// Mitsubishi GX Works2 project: carwash_Q02H_v1   PLC: Q02/Q02H

PROGRAM MAIN
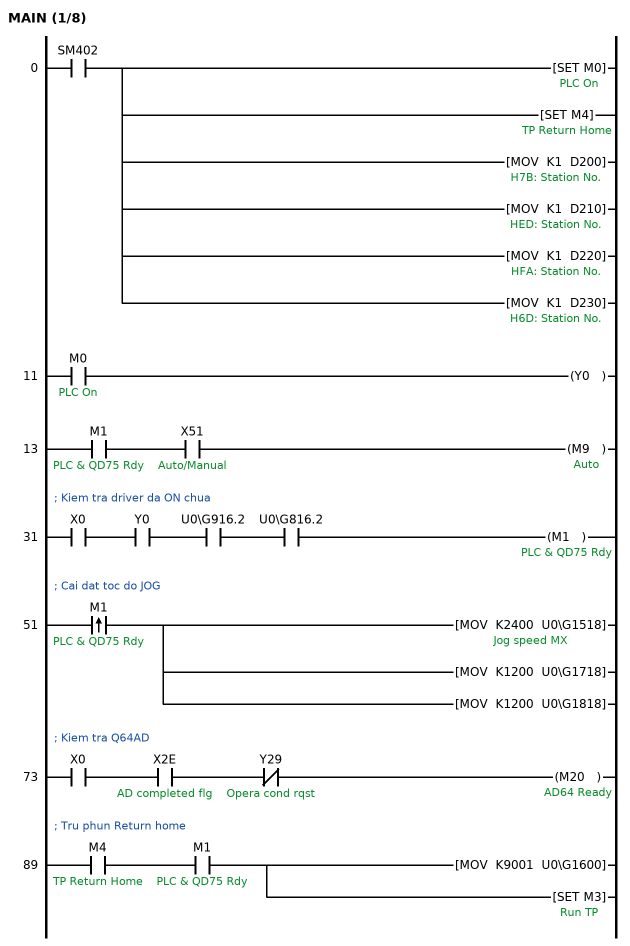
0     LD      SM402
      SET     M0  ; PLC On
      SET     M4  ; TP Return Home
      MOV     K1 D200  ; H7B: Station No.
      MOV     K1 D210  ; HED: Station No.
      MOV     K1 D220  ; HFA: Station No.
      MOV     K1 D230  ; H6D: Station No.
11    LD      M0  ; PLC On
      OUT     Y0
13    LD      M1  ; PLC & QD75 Rdy
      AND     X51  ; Auto/Manual
      OUT     M9  ; Auto
; Kiem tra driver da ON chua
31    LD      X0
      AND     Y0
      AND     U0\G916.2
      AND     U0\G816.2
      OUT     M1  ; PLC & QD75 Rdy
; Cai dat toc do JOG
51    LDP     M1  ; PLC & QD75 Rdy
      MOV     K2400 U0\G1518  ; Jog speed MX
      MOV     K1200 U0\G1718
      MOV     K1200 U0\G1818
; Kiem tra Q64AD
73    LD      X0
      AND     X2E  ; AD completed flg
      ANI     Y29  ; Opera cond rqst
      OUT     M20  ; AD64 Ready
; Tru phun Return home
89    LD      M4  ; TP Return Home
      AND     M1  ; PLC & QD75 Rdy
      MOV     K9001 U0\G1600
      SET     M3  ; Run TP
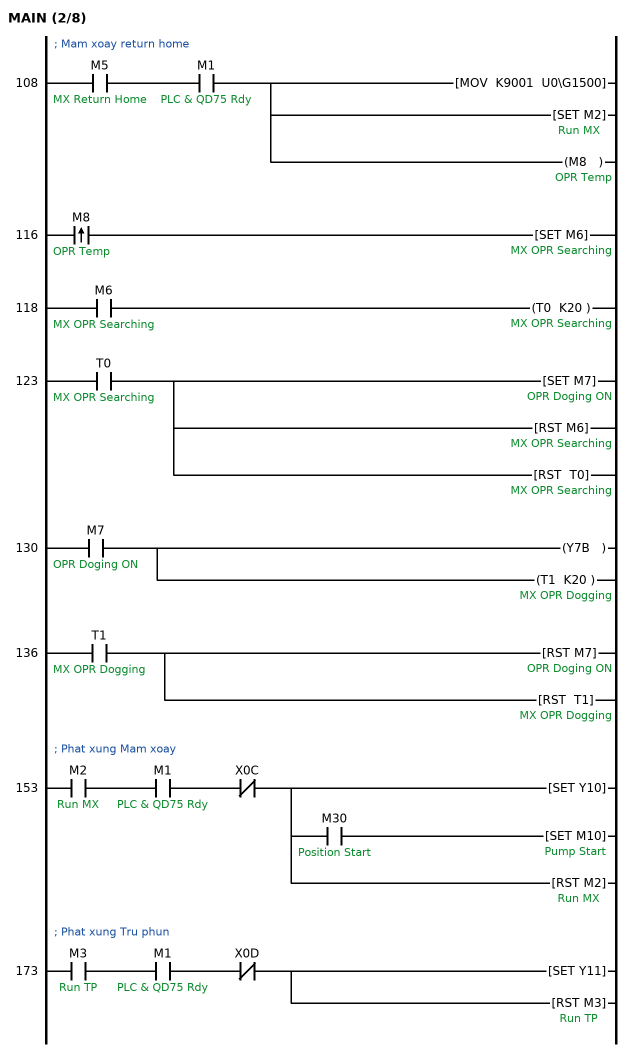
; Mam xoay return home
108   LD      M5  ; MX Return Home
      AND     M1  ; PLC & QD75 Rdy
      MOV     K9001 U0\G1500
      SET     M2  ; Run MX
      OUT     M8  ; OPR Temp
116   LDP     M8  ; OPR Temp
      SET     M6  ; MX OPR Searching
118   LD      M6  ; MX OPR Searching
      OUT     T0 K20  ; MX OPR Searching
123   LD      T0  ; MX OPR Searching
      SET     M7  ; OPR Doging ON
      RST     M6  ; MX OPR Searching
      RST     T0  ; MX OPR Searching
130   LD      M7  ; OPR Doging ON
      OUT     Y7B
      OUT     T1 K20  ; MX OPR Dogging
136   LD      T1  ; MX OPR Dogging
      RST     M7  ; OPR Doging ON
      RST     T1  ; MX OPR Dogging
; Phat xung Mam xoay
153   LD      M2  ; Run MX
      AND     M1  ; PLC & QD75 Rdy
      ANI     X0C
      SET     Y10
      MPS
      AND     M30  ; Position Start
      SET     M10  ; Pump Start
      MPP
      RST     M2  ; Run MX
; Phat xung Tru phun
173   LD      M3  ; Run TP
      AND     M1  ; PLC & QD75 Rdy
      ANI     X0D
      SET     Y11
      RST     M3  ; Run TP
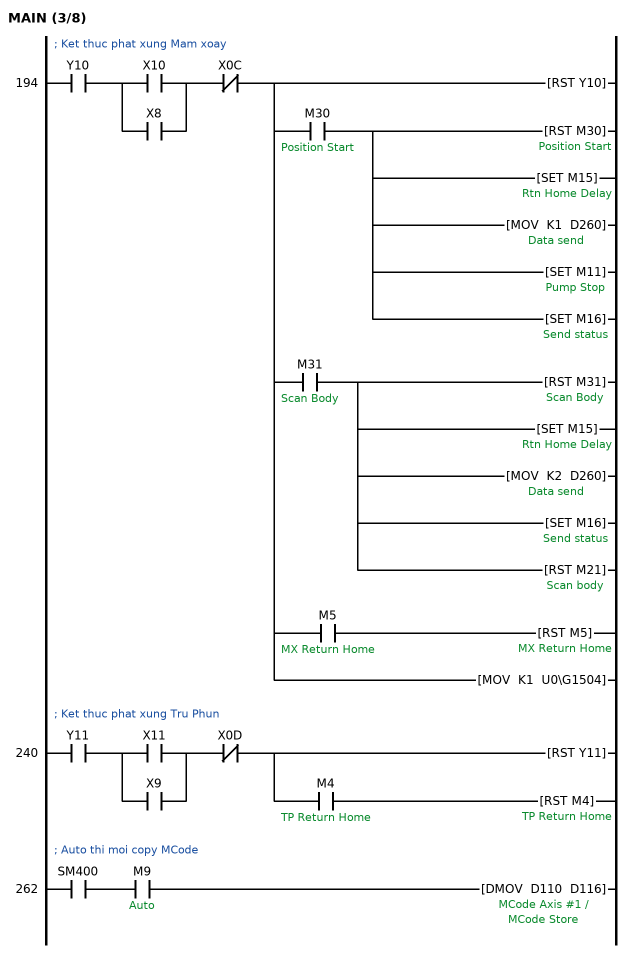
; Ket thuc phat xung Mam xoay
194   LD      Y10
      LD      X10
      OR      X8
      ANB
      ANI     X0C
      RST     Y10
      MPS
      AND     M30  ; Position Start
      RST     M30  ; Position Start
      SET     M15  ; Rtn Home Delay
      MOV     K1 D260  ; Data send
      SET     M11  ; Pump Stop
      SET     M16  ; Send status
      MRD
      AND     M31  ; Scan Body
      RST     M31  ; Scan Body
      SET     M15  ; Rtn Home Delay
      MOV     K2 D260
      SET     M16  ; Send status
      RST     M21  ; Scan body
      MRD
      AND     M5  ; MX Return Home
      RST     M5  ; MX Return Home
      MPP
      MOV     K1 U0\G1504
; Ket thuc phat xung Tru Phun
240   LD      Y11
      LD      X11
      OR      X9
      ANB
      ANI     X0D
      RST     Y11
      AND     M4  ; TP Return Home
      RST     M4  ; TP Return Home
; Auto thi moi copy MCode
262   LD      SM400
      AND     M9  ; Auto
      DMOV    D110 D116  ; MCode Axis #1 / MCode Store
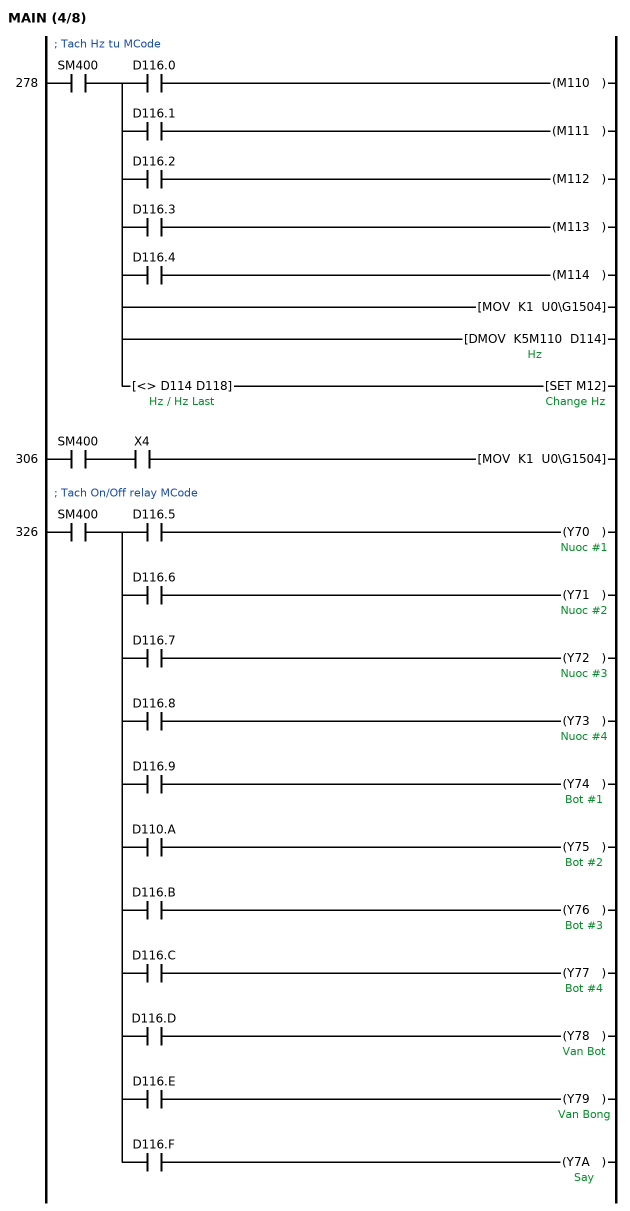
; Tach Hz tu MCode
278   LD      SM400
      MPS
      AND     D116.0
      OUT     M110
      MRD
      AND     D116.1
      OUT     M111
      MRD
      AND     D116.2
      OUT     M112
      MRD
      AND     D116.3
      OUT     M113
      MRD
      AND     D116.4
      OUT     M114
      MPP
      MOV     K1 U0\G1504
      DMOV    K5M110 D114  ; Hz
      AND<>   D114 D118  ; Hz / Hz Last
      SET     M12  ; Change Hz
306   LD      SM400
      AND     X4
      MOV     K1 U0\G1504
; Tach On/Off relay MCode
326   LD      SM400
      MPS
      AND     D116.5
      OUT     Y70  ; Nuoc #1
      MRD
      AND     D116.6
      OUT     Y71  ; Nuoc #2
      MRD
      AND     D116.7
      OUT     Y72  ; Nuoc #3
      MRD
      AND     D116.8
      OUT     Y73  ; Nuoc #4
      MRD
      AND     D116.9
      OUT     Y74  ; Bot #1
      MRD
      AND     D110.A
      OUT     Y75  ; Bot #2
      MRD
      AND     D116.B
      OUT     Y76  ; Bot #3
      MRD
      AND     D116.C
      OUT     Y77  ; Bot #4
      MRD
      AND     D116.D
      OUT     Y78  ; Van Bot
      MRD
      AND     D116.E
      OUT     Y79  ; Van Bong
      MPP
      AND     D116.F
      OUT     Y7A  ; Say
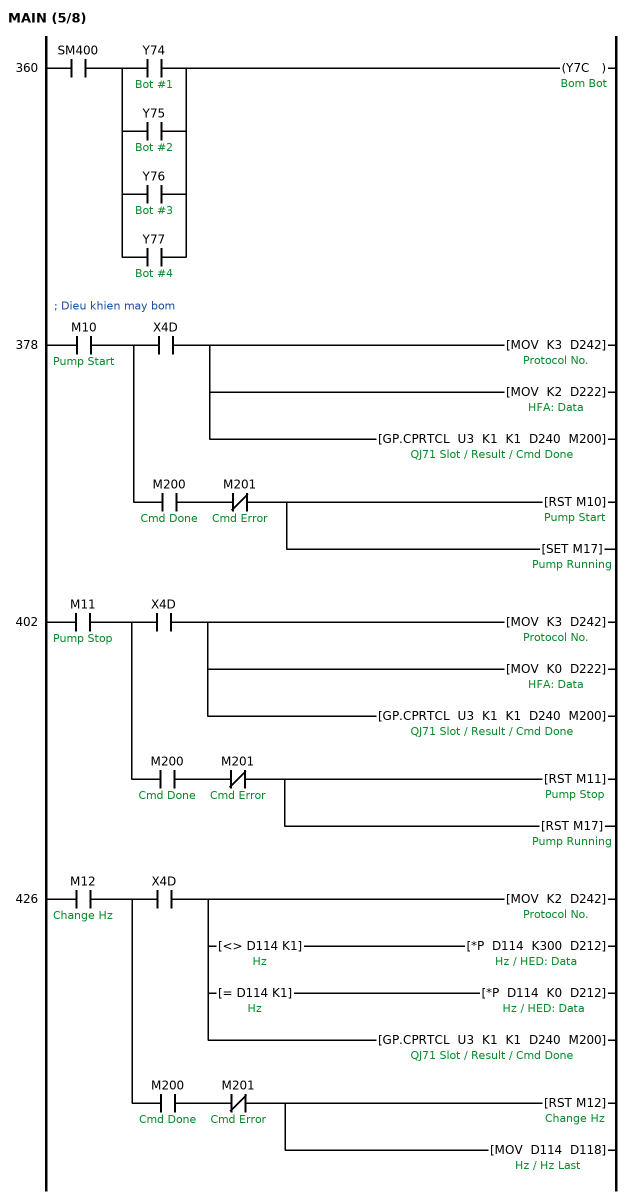
360   LD      SM400
      LD      Y74  ; Bot #1
      OR      Y75  ; Bot #2
      OR      Y76  ; Bot #3
      OR      Y77  ; Bot #4
      ANB
      OUT     Y7C  ; Bom Bot
; Dieu khien may bom
378   LD      M10  ; Pump Start
      MPS
      AND     X4D
      MOV     K3 D242  ; Protocol No.
      MOV     K2 D222  ; HFA: Data
      GP.CPRTCL U3 K1 K1 D240 M200  ; QJ71 Slot / Result / Cmd Done
      MPP
      AND     M200  ; Cmd Done
      ANI     M201  ; Cmd Error
      RST     M10  ; Pump Start
      SET     M17  ; Pump Running
402   LD      M11  ; Pump Stop
      MPS
      AND     X4D
      MOV     K3 D242
      MOV     K0 D222
      GP.CPRTCL U3 K1 K1 D240 M200
      MPP
      AND     M200  ; Cmd Done
      ANI     M201  ; Cmd Error
      RST     M11  ; Pump Stop
      RST     M17  ; Pump Running
426   LD      M12  ; Change Hz
      MPS
      AND     X4D
      MOV     K2 D242
      MPS
      AND<>   D114 K1  ; Hz
      *P      D114 K300 D212  ; HED: Data
      MRD
      AND=    D114 K1  ; Hz
      *P      D114 K0 D212
      MPP
      GP.CPRTCL U3 K1 K1 D240 M200
      MPP
      AND     M200  ; Cmd Done
      ANI     M201  ; Cmd Error
      RST     M12  ; Change Hz
      MOV     D114 D118
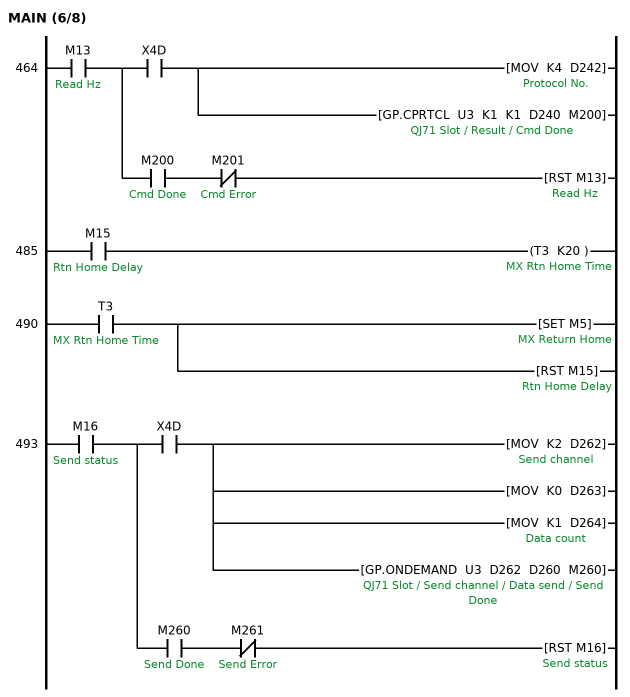
464   LD      M13  ; Read Hz
      MPS
      AND     X4D
      MOV     K4 D242
      GP.CPRTCL U3 K1 K1 D240 M200
      MPP
      AND     M200  ; Cmd Done
      ANI     M201  ; Cmd Error
      RST     M13  ; Read Hz
485   LD      M15  ; Rtn Home Delay
      OUT     T3 K20  ; MX Rtn Home Time
490   LD      T3  ; MX Rtn Home Time
      SET     M5  ; MX Return Home
      RST     M15  ; Rtn Home Delay
493   LD      M16  ; Send status
      MPS
      AND     X4D
      MOV     K2 D262  ; Send channel
      MOV     K0 D263
      MOV     K1 D264  ; Data count
      GP.ONDEMAND U3 D262 D260 M260  ; Send Done
      MPP
      AND     M260  ; Send Done
      ANI     M261  ; Send Error
      RST     M16  ; Send status
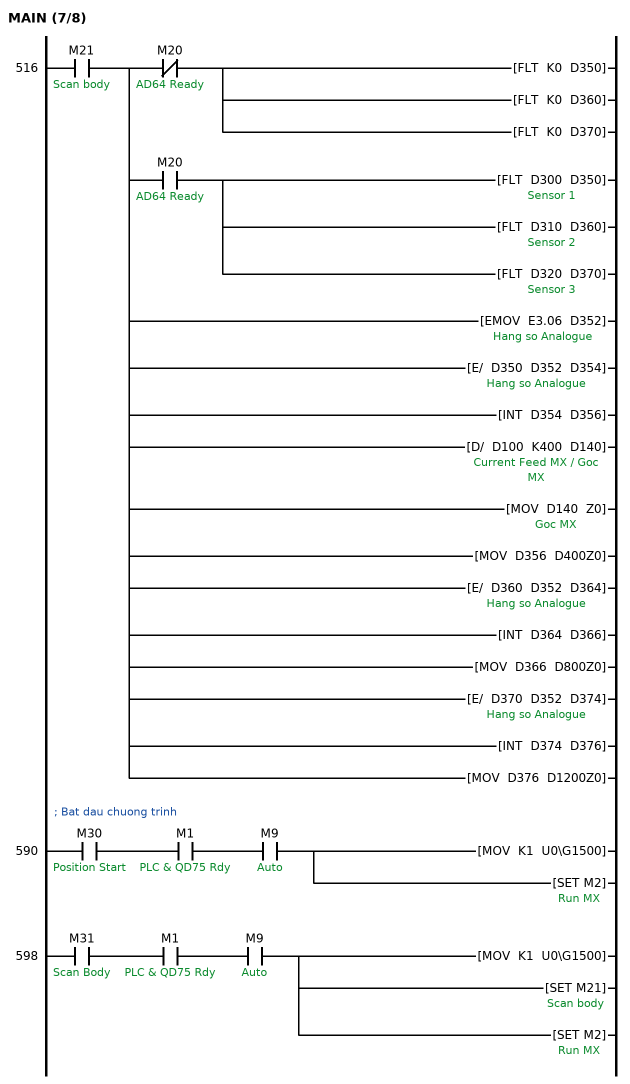
516   LD      M21  ; Scan body
      MPS
      ANI     M20  ; AD64 Ready
      FLT     K0 D350
      FLT     K0 D360
      FLT     K0 D370
      MRD
      AND     M20  ; AD64 Ready
      FLT     D300 D350  ; Sensor 1
      FLT     D310 D360  ; Sensor 2
      FLT     D320 D370  ; Sensor 3
      MPP
      EMOV    E3.06 D352  ; Hang so Analogue
      E/      D350 D352 D354
      INT     D354 D356
      D/      D100 K400 D140  ; Current Feed MX / Goc MX
      MOV     D140 Z0
      MOV     D356 D400Z0
      E/      D360 D352 D364
      INT     D364 D366
      MOV     D366 D800Z0
      E/      D370 D352 D374
      INT     D374 D376
      MOV     D376 D1200Z0
; Bat dau chuong trinh
590   LD      M30  ; Position Start
      AND     M1  ; PLC & QD75 Rdy
      AND     M9  ; Auto
      MOV     K1 U0\G1500
      SET     M2  ; Run MX
598   LD      M31  ; Scan Body
      AND     M1  ; PLC & QD75 Rdy
      AND     M9  ; Auto
      MOV     K1 U0\G1500
      SET     M21  ; Scan body
      SET     M2  ; Run MX
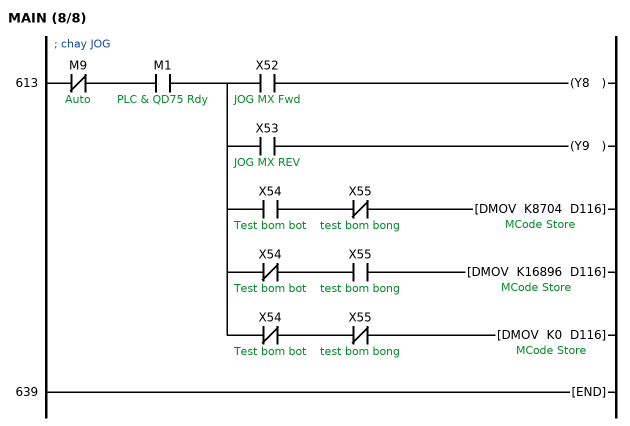
; chay JOG
613   LDI     M9  ; Auto
      AND     M1  ; PLC & QD75 Rdy
      MPS
      AND     X52  ; JOG MX Fwd
      OUT     Y8
      MRD
      AND     X53  ; JOG MX REV
      OUT     Y9
      MRD
      AND     X54  ; Test bom bot
      ANI     X55  ; test bom bong
      DMOV    K8704 D116
      MRD
      ANI     X54  ; Test bom bot
      AND     X55  ; test bom bong
      DMOV    K16896 D116
      MPP
      ANI     X54  ; Test bom bot
      ANI     X55  ; test bom bong
      DMOV    K0 D116
639   END
END_PROGRAM
